(* PLC project Unnamed, Unknown Unnamed 1 *)
(* stored: creationDateTime 2026-06-01T17:35:33, modificationDateTime 2026-06-01T17:35:33 *)

PROGRAM main
  VAR
    bt_start_t1 AT %IX0.0 : BOOL;
    bt_stop_t1 AT %IX0.1 : BOOL;
    bt_emerg_t1 AT %IX0.2 : BOOL;
    led_start_t1 AT %QX0.0 : BOOL;
    led_stop_t1 AT %QX0.1 : BOOL;
    nivel_t1 AT %IW0 : INT;
    vazao_t1 AT %IW1 : INT;
    valv_entrada_t1 AT %QW0 : INT;
    valv_saida_t1 AT %QW1 : INT;
    display_t1 AT %QW2 : INT;
    bt_start_t2 AT %IX0.4 : BOOL;
    bt_stop_t2 AT %IX0.5 : BOOL;
    bt_emerg_t2 AT %IX0.6 : BOOL;
    led_start_t2 AT %QX0.2 : BOOL;
    nivel_t2 AT %IW4 : INT;
    valv_entrada_t2 AT %QW4 : INT;
    valv_saida_t2 AT %QW5 : INT;
    display_t2 AT %QW6 : INT;
    cmd_fill_t1 AT %QX2.0 : BOOL;
    cmd_drain_t1 AT %QX2.1 : BOOL := 0;
    cmd_fill_t2 AT %QX2.2 : BOOL;
    cmd_drain_t2 AT %QX2.3 : BOOL := 0;
    cmd_remote AT %QX2.4 : BOOL;
  END_VAR
  VAR
    mem_start_t1 : BOOL;
    mem_start_t2 : BOOL;
    flag_val_t1 : BOOL;
    flag_val_t2 : BOOL;
    flag_drain_t1 : BOOL;
    flag_drain_t2 : BOOL;
  END_VAR

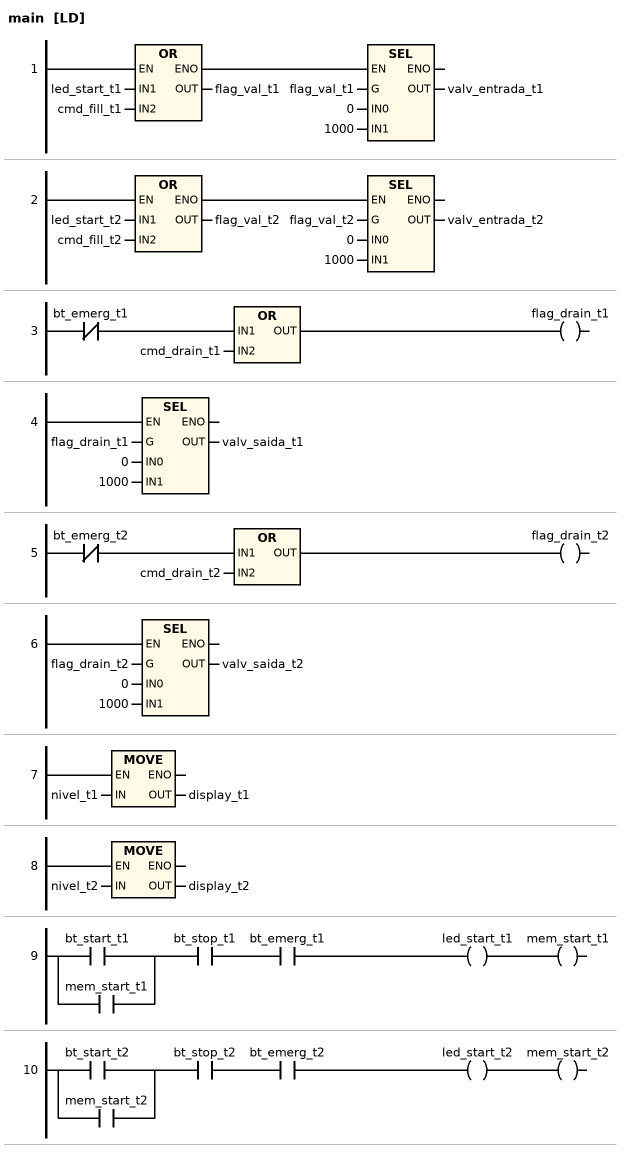
(* LD diagram, written out as Structured Text *)
led_start_t1 := (bt_start_t1 OR mem_start_t1) AND bt_stop_t1 AND bt_emerg_t1;
mem_start_t1 := (bt_start_t1 OR mem_start_t1) AND bt_stop_t1 AND bt_emerg_t1;
led_start_t2 := (bt_start_t2 OR mem_start_t2) AND bt_stop_t2 AND bt_emerg_t2;
mem_start_t2 := (bt_start_t2 OR mem_start_t2) AND bt_stop_t2 AND bt_emerg_t2;
flag_drain_t1 := NOT bt_emerg_t1 OR cmd_drain_t1;
flag_drain_t2 := NOT bt_emerg_t2 OR cmd_drain_t2;
flag_val_t1 := led_start_t1 OR cmd_fill_t1;
valv_entrada_t1 := SEL(flag_val_t1, 0, 1000);
flag_val_t2 := led_start_t2 OR cmd_fill_t2;
valv_entrada_t2 := SEL(flag_val_t2, 0, 1000);
valv_saida_t1 := SEL(flag_drain_t1, 0, 1000);
valv_saida_t2 := SEL(flag_drain_t2, 0, 1000);
display_t1 := nivel_t1;
display_t2 := nivel_t2;
END_PROGRAM

CONFIGURATION Config0
  RESOURCE Res0 ON PLC
    TASK task0(INTERVAL := T#20ms, PRIORITY := 1);
    PROGRAM instance0 WITH task0 : main;
  END_RESOURCE
END_CONFIGURATION
